(* CODESYS project OSC_MQTT.library
   Author: Peter Magnusson
   Title: MQTT Library
   Version: 1.0.0.0
   Description: Open Source CODESYS (OSC) MQTT Client library
   DefaultNamespace: OSC_MQTT
   Company: OSC

Project tree, tasks and I/O mapping:
  libraries: CmpErrors Interfaces, * (System); SysTypes Interfaces, * (System); CmpLog, 3.5.5.0 (System); Standard, 3.5.7.0 (System); CAA Types Extern, 3.5.5.0 (CAA Technical Workgroup); IoStandard, 3.5.8.0 (System); SysMem, 3.5.5.0 (System); CAA Net Base Services, 3.5.8.0 (CAA Technical Workgroup); SysTarget, 3.5.5.0 (System); CmpEventMgr, 3.5.8.0 (System); CmpApp, 3.5.8.0 (System); IoDriver Interfaces, 3.5.2.0 (System); IoDrvBase, 3.5.5.0 (System); IoDriver Parameter Interfaces, 3.5.2.0 (System); SysCpuHandling, 3.5.8.0 (System)
  MQTT/
    Enums/
      data type CLIENTSTATE
      data type MESSAGETYPE
      data type QoS
    Structs/
      data type MQTTMESSAGE
    Function Blocks/
      function block MQTTClient [ST]: _writeByte, _connect, _write, _writeString, _writeWord, _disconnect, Publish, Subscribe, _Send, _Receive, _Keepalive, Initialize
      function block MQTTPub [ST]
      function block IoDrvMQTT [ST]: FB_Init, QueryInterface, FB_Reinit, FB_Exit, Initialize, IoDrvUpdateConfiguration, IoDrvWatchdogTrigger, IoDrvGetModuleDiagnosis, IoDrvStartBusCycle, IoDrvReadInputs, IoDrvUpdateMapping, IoDrvWriteOutputs, IoDrvScanModules, IoDrvIdentify, IoDrvGetConnector, IoDrvWriteParameter, IoDrvReadParameter
    GlobalConstants/
      global variables Constants
*)

// MQTT/Enums/CLIENTSTATE
TYPE CLIENTSTATE :
(
	STOP:= 0,
	INIT,
	CONNECTING,
	CONNECTED,
	DISCONNECTING,
	DISCONNECTED,
	CLOSE,
	ERROR
);
END_TYPE

// MQTT/Enums/MESSAGETYPE
TYPE MESSAGETYPE :
(
	CONNECT 	:= 16#10,
	CONNACK 	:= 16#20,
	PUBLISH 	:= 16#30,
	PUBACK 		:= 16#40,
	SUBSCRIBE 	:= 16#80,
	SUBACK 		:= 16#90,
	UNSUBSCRIBE := 16#A0,
	UNSUBACK 	:= 16#B1,
	PINGREQ 	:= 16#C0,
	PINGRESP	:= 16#D0,
	DISCONNECT 	:= 16#E0
) BYTE;
END_TYPE

// MQTT/Enums/QoS
TYPE QoS :
(
	AtMostOnce:= 2#000,
	AtLeastOnce:= 2#010,
	ExactlyOnce:= 2#100
) BYTE;
END_TYPE

// MQTT/Structs/MQTTMESSAGE
TYPE MQTTMESSAGE :
STRUCT
	MessageType: MESSAGETYPE;
	DUP: BYTE;
	QoS: QoS;
	RetainMsg: BYTE;
	Length: BYTE;
	Payload: ARRAY[0..126] OF BYTE;
END_STRUCT
END_TYPE

// MQTT/GlobalConstants/Constants
{attribute 'qualified_only'}
VAR_GLOBAL CONSTANT	
	MQTTPROTOCOLVERSION : BYTE := BYTE#3;
	MQTT_MAX_PACKET_SIZE : BYTE := 128; //maximum packet size
	
	MQTT_MIN_KEEPALIVE : TIME := T#15S;	
	MQTT_DEFAULT_PORT : UINT := 1883;
	MQTT_MAX_CALLBACKS : INT :=3;
END_VAR

// MQTT/Function Blocks/MQTTClient
FUNCTION_BLOCK MQTTClient
VAR_INPUT
	
END_VAR
VAR_OUTPUT
	xOnline: BOOL;
	dwError: DWORD;

END_VAR
VAR
	sServerIP: STRING;
	uiPort: UINT := 1883;
	tKeepaliveInterval: TIME := T#15S;
	xEnable: BOOL;
	
	MQTT_TIMEAHEAD: TIME;
	Keepalive: TON;
	xKeepaliveEnabled: BOOL;
	xServerAlive:BOOL;

	TCPIPAddress: NBS.IP_ADDR;
	TCPClient: NBS.TCP_Client; /// FB TCP Client 
	TCPConnection: CAA.HANDLE; /// Handle to the established connection 
	TCPRead			: NBS.TCP_Read; (* FB TCP Read *)
	TCPWrite		: NBS.TCP_Write; (* FB TCP Writer *)
	RBUF: ARRAY[0..Constants.MQTT_MAX_PACKET_SIZE] OF BYTE; /// Receive Buffer
	SBUF: ARRAY[0..Constants.MQTT_MAX_PACKET_SIZE] OF BYTE; /// Send Buffer
	sLength: UINT;
	
	_nextMsgId: UINT;
	old_activate: BOOL := FALSE;
	eClientState: CLIENTSTATE;
	ePreviousClientState: CLIENTSTATE;
	cb: BYTE;
	idx1: INT;
	
	_isWriting: MESSAGETYPE; ///Command that is written.
	_hasMessage: BOOL; //has a received message to process
	msgIn: MQTTMESSAGE; //the last received message
	xSend: BOOL;
	_pConnector: POINTER TO IoConfigConnector;
	
END_VAR


Keepalive(IN:=xKeepaliveEnabled, PT:= MQTT_TIMEAHEAD);
//first case of state
IF eClientState <> ePreviousClientState THEN
	CASE eClientState OF
		CLIENTSTATE.INIT:
			{IF defined (DEBUG_MQTTCLIENT)}
			LogAdd(STD_LOGGER,'MQTTClient',UDINT_TO_DINT(LogClass.LOG_INFO),0,0,'State.INIT');
			{END_IF}
			MQTT_TIMEAHEAD:= UDINT_TO_TIME(TIME_TO_UDINT(tKeepaliveInterval) / 3 * 2);// 2/3 to be paranoid 
		CLIENTSTATE.CONNECTING:
			{IF defined (DEBUG_MQTTCLIENT)}
			LogAdd(STD_LOGGER,'MQTTClient',UDINT_TO_DINT(LogClass.LOG_INFO),0,0,'State.CONNECTING');
			{END_IF}
		CLIENTSTATE.CONNECTED:
			{IF defined (DEBUG_MQTTCLIENT)}
			LogAdd(STD_LOGGER,'MQTTClient',UDINT_TO_DINT(LogClass.LOG_INFO),0,0,'State.CONNECTED');
			{END_IF}
		CLIENTSTATE.DISCONNECTING:
			{IF defined (DEBUG_MQTTCLIENT)}
			LogAdd(STD_LOGGER,'MQTTClient',UDINT_TO_DINT(LogClass.LOG_INFO),0,0,'State.DISCONNECTING');
			{END_IF}
		CLIENTSTATE.DISCONNECTED:
			{IF defined (DEBUG_MQTTCLIENT)}
			LogAdd(STD_LOGGER,'MQTTClient',UDINT_TO_DINT(LogClass.LOG_INFO),0,0,'State.DISCONNECTED');
			{END_IF}
		CLIENTSTATE.CLOSE:		
			{IF defined (DEBUG_MQTTCLIENT)}
			LogAdd(STD_LOGGER,'MQTTClient',UDINT_TO_DINT(LogClass.LOG_INFO),0,0,'State.CLOSE');
			{END_IF}
		CLIENTSTATE.ERROR:
			{IF defined (DEBUG_MQTTCLIENT)}
			LogAdd(STD_LOGGER,'MQTTClient',UDINT_TO_DINT(LogClass.LOG_INFO),0,0,'State.ERROR');
			{END_IF}
	END_CASE
END_IF
ePreviousClientState:= eClientState;

//every time the loop is in a certain state.
CASE eClientState OF
	
	CLIENTSTATE.STOP:
		xOnline := FALSE;
		
	CLIENTSTATE.INIT:
		SysMem.SysMemSet(ADR(SBUF), 0, SIZEOF(SBUF)); //clear send buffer;
		SysMem.SysMemSet(ADR(RBUF), 0, SIZEOF(RBUF)); //clear receive buffer;
		TCPIPAddress.sAddr := sServerIP;
		xSend:=FALSE;
		dwError := 0;
		sLength:=0;
		_hasMessage:= FALSE;
		_nextMsgId := 1;
		TCPWrite(xExecute:= FALSE);
		(* The client tries to establish a connection to a mqtt server *)
		TCPClient(xEnable:= TRUE, udiTimeOut:= 0, ipAddr:= TCPIPAddress, uiPort:= uiPort, hConnection=> TCPConnection);
		
			
		IF TCPClient.xActive THEN 
			eClientState:= CLIENTSTATE.CONNECTING;
			xServerAlive:=TRUE;
			THIS^._connect();
		ELSIF TCPClient.xError THEN
			
			eClientState:= CLIENTSTATE.ERROR;
		END_IF	
	(*------------------------- *)
	

	
	CLIENTSTATE.CONNECTED:
			xKeepaliveEnabled:= TRUE;
			xOnline:= TRUE;
	(*------------------------- *)
	
	CLIENTSTATE.DISCONNECTING:
			xKeepaliveEnabled:=FALSE;
			IF NOT xSend THEN
				eClientState:= DISCONNECTED;
			END_IF
	(*------------------------- *)	
	
	CLIENTSTATE.DISCONNECTED:		
		//logger('disconnected');
		xKeepaliveEnabled:=FALSE;
		eClientState:= CLOSE;
	(*------------------------- *)
	
	CLIENTSTATE.ERROR:
		xSend:=FALSE;
		TCPClient(xEnable := FALSE);
		eCLientState:= CLOSE;
		
	(*------------------------- *)
	
	CLIENTSTATE.CLOSE:		
		//logger('close');
		xServerAlive:=FALSE;
		xKeepaliveEnabled:=FALSE;
		old_activate := FALSE;
		xOnline:= FALSE;
		
		TCPWrite(xExecute:= FALSE);
		TCPRead(xEnable:=FALSE);
		TCPClient(xEnable:= FALSE);
		
		eClientState := CLIENTSTATE.STOP;
		
		
		
	(*------------------------- *)
	
END_CASE




//IPC1(IP:= DWORD#0, PORT:= WORD#0 , TIME_OUT:= TIMEOUT, IP_C:= IP_C1, S_BUF:= S_BUF1, R_BUF:= R_BUF1); (* MQTT Connection *)




IF NOT old_activate AND xEnable THEN
	eClientState := INIT;
	old_activate:= TRUE;
END_IF

IF NOT xEnable AND old_activate THEN
	{IF defined (DEBUG_MQTTCLIENT)}
	LogAdd(STD_LOGGER,'MQTTClient',UDINT_TO_DINT(LogClass.LOG_INFO),0,0,'Falling flank of xConnect ');
	{END_IF}
	THIS^._disconnect();
	old_activate:= FALSE;
END_IF

IF xSend AND TCPConnection = CAA.gc_hINVALID THEN
	xSend:= FALSE;
	IF eClientState <= CLIENTSTATE.DISCONNECTED THEN
		eClientState:= CLIENTSTATE.DISCONNECTED;
	END_IF
	
END_IF


IF TCPClient.xEnable AND TCPClient.xActive AND TCPClient.hConnection <> CAA.gc_hINVALID THEN
	THIS^._Keepalive();
	THIS^._Send();
	THIS^._Receive();
END_IF

METHOD PRIVATE _writeByte : INT
VAR_IN_OUT
	pos: UINT;
END_VAR
VAR_INPUT
	b: BYTE;
	pBuf: POINTER TO ARRAY[0..Constants.MQTT_MAX_PACKET_SIZE] OF BYTE;
END_VAR
//Add to current position according to size
pBuf^[pos]:= b;
//increase size
pos:= pos +1;
END_METHOD

METHOD PRIVATE _connect : BOOL
VAR_INPUT

END_VAR
VAR
	name: WSTRING:="01234567890123456789";
	dwId: DWORD;
	id: STRING;
	v: BYTE;
	w: UINT;
	length: UINT;
	MAX_NAME_LENGTH: UDINT := 20;
END_VAR

IF TCPClient.xActive THEN
		
	SysTarget.SysTargetGetNodeName(ADR(name), ADR(MAX_NAME_LENGTH));
	SysTarget.SysTargetGetId(ADR(dwId));
	id := CONCAT('mqttio/', WSTRING_TO_STRING(name));
	id := CONCAT(id, '-');
	id := CONCAT(id, DWORD_TO_STRING(dwId));
	
	 

	// {0x00,0x06,'M','Q','I','s','d','p',MQTTPROTOCOLVERSION};
	//leave room in the buffer for header and variable field length field
	length:=2;
	//start adding
	_writeByte(pos:=length, b:=16#0, pBuf := ADR(SBUF));
	_writeByte(pos:=length, b:=16#6, pBuf := ADR(SBUF));
	_writeString(pos:=length, msg:='MQIsdp');
	_writeByte(pos:=length, b:=Constants.MQTTPROTOCOLVERSION, pBuf := ADR(SBUF));
	
	//connect flags
	v := 16#2;//no will topic
	_writeByte(pos:=length, b:=v, pBuf := ADR(SBUF));
	
	//Keep Alive Timer
	_writeWord(pos:=length, w:= TIME_TO_WORD(tKeepaliveInterval/1000),  pBuf := ADR(SBUF)); 
	
	//client id length
	w:= INT_TO_UINT(LEN(id));
	_writeWord(pos:=length, w:=w,  pBuf := ADR(SBUF));
	//client id
	_writeString(pos:=length, msg:=id);
	_write(MESSAGETYPE.CONNECT, length);

END_IF
END_METHOD

METHOD PRIVATE _write : BOOL
VAR_INPUT
	header: MESSAGETYPE;
	length: UINT;
END_VAR
VAR
	len: BYTE;
END_VAR
IF TCPClient.xActive THEN	
	{IF defined (DEBUG_MQTTCLIENT)}
	LogAdd(STD_LOGGER,'MQTTClient',UDINT_TO_DINT(LogClass.LOG_INFO),0,0,CONCAT('Writing msg:', BYTE_TO_STRING(header) ));
	{END_IF}
	_isWriting:= header;
	len:= UINT_TO_BYTE(length);
	SBUF[0]:= header;
	IF len >= 2 THEN
		SBUF[1]:= len -2;
	ELSE
		SBUF[1]:= 0;
	END_IF
	
	IF(length<2) THEN
		length:= 2;
	END_IF
	sLength:= length;
	xSend:= TRUE;
END_IF
END_METHOD

METHOD PRIVATE _writeString
VAR_IN_OUT
	pos: UINT;
END_VAR
VAR_INPUT
	msg: STRING;
	
END_VAR

VAR
	ps : POINTER TO BYTE;
	end: UINT;
	i: UINT;
	length: UINT;
END_VAR
ps := ADR(msg);
length := INT_TO_UINT(LEN(msg));
end := MIN(pos + length, SIZEOF(SBUF));
IF end > 0 THEN end := end -1; END_IF;
FOR i := pos TO end DO
	SBUF[i] := ps^;
	ps := ps + 1;
END_FOR;
pos:=pos + length;
END_METHOD

METHOD PRIVATE _writeWord : INT
VAR_IN_OUT
	pos: UINT;
END_VAR
VAR_INPUT
	w: WORD;
	pBuf: POINTER TO ARRAY[0..Constants.MQTT_MAX_PACKET_SIZE] OF BYTE;
END_VAR
VAR
	v: BYTE;
	length: UINT;
END_VAR
length:= pos;
v:= UINT_TO_BYTE(SHR(w, 8));
_writeByte(pos:=length, b:=v, pBuf:=pBuf );
v:= UINT_TO_BYTE(w AND 16#FF);
_writeByte(pos:=length, b:=v, pBuf := pBuf); 
pos:= length;
END_METHOD

METHOD PRIVATE _disconnect
VAR_INPUT
END_VAR

VAR
	
END_VAR
{IF defined (DEBUG_MQTTCLIENT)}
LogAdd(STD_LOGGER,'MQTTClient',UDINT_TO_DINT(LogClass.LOG_INFO),0,0,'Calling _Disconnect');
{END_IF}
SysMem.SysMemSet(ADR(SBUF), 0, Constants.MQTT_MAX_PACKET_SIZE); //clear send buffer;
THIS^._write(MESSAGETYPE.DISCONNECT, 0);
eCLIENTSTATE:= CLIENTSTATE.DISCONNECTING;
END_METHOD

METHOD Publish
VAR_INPUT
	sTopic: STRING;
	sValue: STRING;
	xExecute: BOOL;
	bQos: BYTE;
	xRetain:BOOL;
END_VAR
VAR_OUTPUT
	xDone:BOOL;
END_VAR
VAR
	length: UINT;
	xBusyPublishing:BOOL; //will be set if publishing
	bBuf : ARRAY[0..Constants.MQTT_MAX_PACKET_SIZE] OF BYTE; /// Send Buffer
END_VAR

IF xExecute AND NOT xBusyPublishing THEN //Rising flank
	IF TCPClient.xActive THEN
		{IF defined (DEBUG_MQTTCLIENT)}
		LogAdd(STD_LOGGER,'MQTTClient',UDINT_TO_DINT(LogClass.LOG_INFO),0,0,'Publishing');
		{END_IF}
		xDone:=FALSE;
		xBusyPublishing:=TRUE;
		//sTopic := concat(sTopicPrefix, sTopic);
		length:= 2;//starting position in the buffer
		_writeWord(pos:=length, w:= INT_TO_UINT(LEN(sTopic)), pBuf := ADR(bBuf));
		_writeString(pos:=length, msg:=sTopic);
		IF bQos > 0 THEN //only send msg id if needed.
			_writeWord(pos:=length, w:= _nextMsgId, pBuf := ADR(SBUF));
		END_IF
		_writeString(pos:=length, msg:=sValue);
		_write(MESSAGETYPE.PUBLISH, length);
	END_IF
ELSIF NOT xExecute AND xBusyPublishing THEN //falling flank
	{IF defined (DEBUG_MQTTCLIENT)}
	LogAdd(STD_LOGGER,'MQTTClient',UDINT_TO_DINT(LogClass.LOG_INFO),0,0,'Publishing falling');
	{END_IF}
	xDone:=FALSE;
	xBusyPublishing:=FALSE;
ELSIF xExecute AND xBusyPublishing THEN //steady high
	//TODO:Wait for PUBACK if QoS >0
	IF NOT xSend THEN
		{IF defined (DEBUG_MQTTCLIENT)}
		LogAdd(STD_LOGGER,'MQTTClient',UDINT_TO_DINT(LogClass.LOG_INFO),0,0,'Publishing Done');
		{END_IF}
		xDone:=TRUE;
	END_IF
END_IF
END_METHOD

METHOD Subscribe : BOOL
VAR_INPUT
	sTopic: STRING;
	//pfbCallback: POINTER TO IMqttMessage;
END_VAR

VAR
	length: UINT;
END_VAR
//Save callback for later and send subscribe message
//m_Subscriptions.AddSub(sTopic:=sTopic, pfbCallback:=pfbCallback);

//leave room in the buffer for header and variable field length field
length:=2;

//topic and length of topic
_writeWord(pos:=length, INT_TO_UINT(LEN(sTopic)), pBuf := ADR(SBUF));
_writeString(pos:=length, msg:=sTopic);

//requested qos
_writeByte(pos:=length, b:=0, pBuf := ADR(SBUF));

_write(MESSAGETYPE.SUBSCRIBE, length);
END_METHOD

METHOD PRIVATE _Send
VAR_INPUT
END_VAR
IF xSend THEN
	

{IF defined (DEBUG_MQTTCLIENT)}
LogAdd(STD_LOGGER,'MQTTClient',UDINT_TO_DINT(LogClass.LOG_INFO),0,0,'Sending...');
{END_IF}
TCPWrite(xExecute:= TRUE, udiTimeOut:= 0, hConnection:= TCPConnection, szSize:= sLength, pData:= ADR(SBUF));
IF TCPWrite.xDone THEN 
	_nextMsgId:= _nextMsgId +1;				
	TCPWrite(xExecute:= FALSE);	
	xSend:= FALSE;
	sLength:= 0;		
	{IF defined (DEBUG_MQTTCLIENT)}
	LogAdd(STD_LOGGER,'MQTTClient',UDINT_TO_DINT(LogClass.LOG_INFO),0,0,'Sent');
	{END_IF}	
ELSIF TCPWrite.xError THEN
	//eCLIENTSTATE := CLIENTSTATE.ERROR;
	TCPWrite(xExecute:=FALSE);
	xSend:= FALSE;
	sLength:=0;
	{IF defined (DEBUG_MQTTCLIENT)}
	LogAdd(STD_LOGGER,'MQTTClient',UDINT_TO_DINT(LogClass.LOG_INFO),0,0,'Error Sending');
	{END_IF}
END_IF
IF _isWriting = MESSAGETYPE.DISCONNECT THEN
	eClientState := CLIENTSTATE.DISCONNECTED;
	xSend:=FALSE;
	{IF defined (DEBUG_MQTTCLIENT)}
	LogAdd(STD_LOGGER,'MQTTClient',UDINT_TO_DINT(LogClass.LOG_INFO),0,0,'Send Disconnect');
	{END_IF}
END_IF

END_IF
END_METHOD

METHOD PRIVATE _Receive
VAR_INPUT
END_VAR
TCPRead(xEnable:= TRUE, hConnection:= TCPConnection, szSize:= Constants.MQTT_MAX_PACKET_SIZE, pData:= ADR(RBUF));
IF TCPRead.xReady AND TCPRead.szCount > 0 THEN
	msgIn.MessageType := RBUF[0] AND 16#F0; //mask of first half
	msgIn.DUP := RBUF[0] AND 16#08;
	msgIn.QoS := RBUF[0] AND 16#06;
	msgIn.RetainMsg := RBUF[0] AND 1;
	msgIn.Length := RBUF[1]; //remaining length;
	SysMem.SysMemCpy(ADR(msgIn.Payload[0]), ADR(RBUF[2]), msgIn.Length);
	_hasMessage := TRUE;
	{IF defined (DEBUG_MQTTCLIENT)}
	LogAdd(STD_LOGGER,'MQTTClient',UDINT_TO_DINT(LogClass.LOG_INFO),0,0,CONCAT('Received:', BYTE_TO_STRING(msgIn.MessageType)));
	{END_IF}
ELSIF TCPRead.xError THEN
	eClientState := CLIENTSTATE.ERROR;
	{IF defined (DEBUG_MQTTCLIENT)}
	LogAdd(STD_LOGGER,'MQTTClient',UDINT_TO_DINT(LogClass.LOG_INFO),0,0,'Receive Error');
	{END_IF}
END_IF




IF _hasMessage THEN
//logger('hasMessage');	
	CASE _isWriting OF
		MESSAGETYPE.CONNECT:
			IF msgIn.MessageType = MESSAGETYPE.CONNACK THEN
				IF msgIn.Payload[1] = 0 THEN //connection accepted
					eClientState:= CONNECTED; 
					
				ELSE
					{IF defined (DEBUG_MQTTCLIENT)}
					LogAdd(STD_LOGGER,'MQTTClient',UDINT_TO_DINT(LogClass.LOG_INFO),0,0,'Could not authenticate');
					{END_IF}
					eClientState:= CLOSE;	
				END_IF
			END_IF
		(*----------------------------*)
		
		MESSAGETYPE.SUBSCRIBE:
			IF msgIn.MessageType = MESSAGETYPE.SUBACK THEN
				{IF defined (DEBUG_MQTTCLIENT)}
				LogAdd(STD_LOGGER,'MQTTClient',UDINT_TO_DINT(LogClass.LOG_INFO),0,0,'SUBACK');
				{END_IF}
			ELSE
				{IF defined (DEBUG_MQTTCLIENT)}
				LogAdd(STD_LOGGER,'MQTTClient',UDINT_TO_DINT(LogClass.LOG_INFO),0,0,'SUBACK EXPECTED BUT NOT RECEIVED');
				{END_IF}	
			END_IF
			
		(*----------------------------*)
		
		MESSAGETYPE.PINGREQ:
			IF msgIn.MessageType = MESSAGETYPE.PINGRESP THEN
				//server alive
				{IF defined (DEBUG_MQTTCLIENT)}
				LogAdd(STD_LOGGER,'MQTTClient',UDINT_TO_DINT(LogClass.LOG_INFO),0,0,'PINGRESP');
				{END_IF}
				xServerAlive:=TRUE;
			END_IF 
		(*----------------------------*)
		
	
	END_CASE
_hasMessage:= FALSE; //message is dealt with
END_IF
END_METHOD

METHOD PRIVATE _Keepalive
VAR_INPUT
END_VAR
//keepalive triggered
IF Keepalive.Q THEN
	xKeepaliveEnabled:= FALSE;
	IF NOT xServerAlive THEN
		//SOMETHING BAD HAPPENED
		{IF defined (DEBUG_MQTTCLIENT)}
		LogAdd(STD_LOGGER,'MQTTClient',UDINT_TO_DINT(LogClass.LOG_INFO),0,0,'Something bad happened with connection');
		{END_IF}
		eClientState:= CLOSE;
	ELSE
		//check if server is alive.
		xServerAlive:=FALSE;
		{IF defined (DEBUG_MQTTCLIENT)}
		LogAdd(STD_LOGGER,'MQTTClient',UDINT_TO_DINT(LogClass.LOG_INFO),0,0,'PINGREQ');
		{END_IF}
		_write(MESSAGETYPE.PINGREQ, 0);
	END_IF
END_IF
END_METHOD

METHOD Initialize : UDINT
VAR_INPUT
	wModuleType : UINT;
	dwInstance : UDINT;
	pConnector : POINTER TO IoConfigConnector;
END_VAR
VAR
	pParam: POINTER TO IoConfigParameter;		
	udiResult: UDINT;
END_VAR

pParam := ConfigGetParameter(_pConnector, 1);
IF pParam <> 0 THEN
	_byHardwareAddress := IoStandard.ConfigGetParameter(pParam, ADR(udiResult));
END_IF
END_METHOD

END_FUNCTION_BLOCK

// MQTT/Function Blocks/MQTTPub
FUNCTION_BLOCK MQTTPub
VAR_INPUT
	pClient		:POINTER TO MQTTClient;
	sTopic		:STRING;
	sValue		:STRING;
	xExecute	:BOOL;
END_VAR
	
VAR_OUTPUT
	xDone		:BOOL;
END_VAR
VAR
	
END_VAR

IF xExecute THEN
	pClient^.Publish(sTopic:=sTopic, sValue:=sValue, bQos:=0, xRetain:=FALSE, xExecute:=TRUE, xDone => xDone);
END_IF

END_FUNCTION_BLOCK

// MQTT/Function Blocks/IoDrvMQTT
FUNCTION_BLOCK IoDrvMQTT EXTENDS IoDrvBase IMPLEMENTS ICmpIoDrvParameter
VAR_INPUT
END_VAR
VAR_OUTPUT
	
END_VAR
VAR CONSTANT
	CLASSID_CCmpIoDrvTemplate : DWORD := 16#0000FF02; //TODO
	_IIoDrv : ICmpIoDrv;
	_IIoDrvParameter : ICmpIoDrvParameter;
	_xBackGroundDiagStarted : BOOL;
	_bDeactivated : BOOL;
	Client: MQTTClient;
END_VAR

VAR
END_VAR

{attribute 'conditionalshow'}
METHOD FB_Init : BOOL
VAR_INPUT
	bInitRetains	: BOOL;
	bInCopyCode	: BOOL;
END_VAR
VAR
	Result : UDINT;
END_VAR
FB_Init_Count := FB_Init_Count + 1;

m_Info.szDriverName := 'IoDrvMQTT';
m_Info.szVendorName := 'Open Source CODESYS (OSC)';
m_Info.szDeviceName := 'MQTT';
m_Info.wModuleType := 501;

_IIoDrv := THIS^;
_IIoDrvParameter := THIS^;

m_IBaseItf := THIS^;
m_hInterface := IoMgrRegisterInstance2(CLASSID_CCmpIoDrvTemplate, m_IBaseItf, ADR(Result));
FB_Init := TRUE;
END_METHOD

{attribute 'conditionalshow'}
METHOD QueryInterface : POINTER TO POINTER TO BYTE
VAR_INPUT
	(* InterfaceID *)
	iid	: DWORD;
	pResult	: POINTER TO UDINT;
END_VAR
QueryInterface_Count := QueryInterface_Count + 1;
IF iid = ITFID_ICmpIoDrv THEN
	QueryInterface := ADR(_IIoDrv);
	AddRef();
	IF (pResult <> 0) THEN
		pResult^ := Errors.ERR_OK;
	END_IF
	RETURN;	
ELSIF iid = ITFID_ICmpIoDrvParameter THEN
	QueryInterface := ADR(_IIoDrvParameter);
	AddRef();
	IF (pResult <> 0) THEN
		pResult^ := Errors.ERR_OK;
	END_IF	
	RETURN;	
ELSE
	QueryInterface := SUPER^.QueryInterface(iid, pResult);
END_IF
END_METHOD

{attribute 'conditionalshow'}
METHOD FB_Reinit : BOOL
FB_Reinit_Count := FB_Reinit_Count + 1;
FB_Reinit := TRUE;
END_METHOD

{attribute 'conditionalshow'}
METHOD FB_Exit : BOOL
VAR_INPUT
	bInCopyCode	: BOOL;
END_VAR
FB_Exit_Count := FB_Exit_Count + 1;
FB_Exit := TRUE;
END_METHOD

{attribute 'conditionalshow'}
METHOD Initialize : UDINT
VAR_INPUT
	wModuleType : UINT;
	dwInstance : UDINT;
	pConnector : POINTER TO IoConfigConnector; 
END_VAR
Initialize_Count := Initialize_Count + 1;

m_wModuleType := wModuleType;
m_dwInstance := dwInstance;
m_Info.wModuleType := wModuleType;

Client.Initialize(wModuleType, dwInstance, pConnector);

Initialize := Errors.ERR_OK;
END_METHOD

{attribute 'conditionalshow'}
METHOD IoDrvUpdateConfiguration : UDINT
VAR_INPUT
	pConnectorList	: POINTER TO IoConfigConnector;
	nCount	: DINT;
END_VAR

VAR
	pParameter : POINTER TO IoConfigParameter;	
	pChild : POINTER TO IoConfigConnector;	
	pstConnectorVendorName : POINTER TO STRING;
	pstConnectorDeviceName : POINTER TO STRING;
	dwTest : POINTER TO DWORD;
	Result : RTS_IEC_RESULT;
END_VAR
IoDrvUpdateConfiguration_Count := IoDrvUpdateConfiguration_Count + 1;
IoDrvUpdateConfiguration := Errors.ERR_OK;

IF (pConnectorList = 0) THEN
	// Reset application
	// TODO: Free ressources
	RETURN;
END_IF

m_pConnector := IoMgrConfigGetConnector(pConnectorList, ADR(nCount), m_wModuleType, m_dwInstance);

IF m_pConnector = 0 THEN
	IoDrvUpdateConfiguration := ERRORS.ERR_PARAMETER;
	RETURN;
END_IF

//check if device is enabled in the device tree
IF (m_pConnector^.dwFlags AND ConnectorFlags.CF_ENABLE) = 0 THEN
	_bDeactivated := TRUE;
	IoDrvUpdateConfiguration := Errors.ERR_OK;
	RETURN;
END_IF

IF m_pConnector^.hIoDrv = 0 THEN
	m_pConnector^.hIoDrv := m_hInterface;
	m_pConnector^.pFather^.hIoDrv := m_hInterface;
	
	{IF defined (pou:IoMgrConfigSetDiagnosis)}
	IoMgrConfigSetDiagnosis(m_pConnector,
							ConnectorFlags.CF_DRIVER_AVAILABLE OR
							ConnectorFlags.CF_CONNECTOR_FOUND OR
							ConnectorFlags.CF_CONNECTOR_CONFIGURED OR
							ConnectorFlags.CF_CONNECTOR_ACTIVE);
	{END_IF}
	
	{IF defined (pou:IoMgrConfigSetDiagnosis)}
	IoMgrConfigSetDiagnosis(m_pConnector^.pFather,
							ConnectorFlags.CF_DRIVER_AVAILABLE OR
							ConnectorFlags.CF_CONNECTOR_FOUND OR
							ConnectorFlags.CF_CONNECTOR_CONFIGURED OR
							ConnectorFlags.CF_CONNECTOR_ACTIVE);
	{END_IF}

	{IF defined (pou:IoMgrSetDriverProperties)}			
		IoMgrSetDriverProperties(m_hInterface, DRVPROP_CONSISTENCY OR DRVPROP_BACKGROUND_GETDIAG);
		//Note: background diagnosis property flag is optional (supported with 3.5.1.0 runtime)
	{END_IF}										

	//Setup I/O area
	pParameter := IoMgrConfigGetParameter(m_pConnector, 1000);		(* inputs *)
	IF (pParameter <> 0) THEN
		pParameter^.dwDriverSpecific := 0;					(* Device offset 0 *)
	END_IF
	pParameter := IoMgrConfigGetParameter(m_pConnector, 2000);		(* outputs *)
	IF (pParameter <> 0) THEN
		pParameter^.dwDriverSpecific := 0;					(* Device offset 0 *)
	END_IF
	
	//Go through all childs of the device
	pChild := IoMgrConfigGetFirstChild(m_pConnector, ADR(nCount), m_pConnector);
	WHILE (pChild <> 0) DO
		IF (pChild^.dwFlags AND ConnectorFlags.CF_ENABLE) <> 0 THEN
			pChild^.hIoDrv := m_hInterface;	
			{IF defined (pou:IoMgrConfigSetDiagnosis)}
			IoMgrConfigSetDiagnosis(pChild,
									ConnectorFlags.CF_DRIVER_AVAILABLE OR
									ConnectorFlags.CF_CONNECTOR_FOUND OR
									ConnectorFlags.CF_CONNECTOR_CONFIGURED OR
									ConnectorFlags.CF_CONNECTOR_ACTIVE);
			{END_IF}
		END_IF
		pChild := IoMgrConfigGetNextChild(pChild, ADR(nCount), m_pConnector);
	END_WHILE
END_IF
END_METHOD

{attribute 'conditionalshow'}
METHOD IoDrvWatchdogTrigger : UDINT
VAR_INPUT
	pConnector	: POINTER TO IoConfigConnector;
END_VAR
IoDrvWatchdogTrigger_Count := IoDrvWatchdogTrigger_Count + 1;
IoDrvWatchdogTrigger := Errors.ERR_OK;
END_METHOD

{attribute 'conditionalshow'}
METHOD IoDrvGetModuleDiagnosis : UDINT
VAR_INPUT
	pConnector	: POINTER TO IoConfigConnector;
END_VAR
IF pConnector = 0 THEN
	//we are called from the background task
	_xBackGroundDiagStarted := TRUE;
END_IF

//Todo: update connectorflags if something changed

IoDrvGetModuleDiagnosis_Count := IoDrvGetModuleDiagnosis_Count + 1;
IoDrvGetModuleDiagnosis := Errors.ERR_NOTIMPLEMENTED;
END_METHOD

{attribute 'conditionalshow'}
METHOD IoDrvStartBusCycle : UDINT
VAR_INPUT
	pConnector	: POINTER TO IoConfigConnector;
END_VAR
IoDrvStartBusCycle_Count := IoDrvStartBusCycle_Count + 1;

//if background diagnosis is not active call IoDrvGetModuleDiagnosis; normally it will be called by the runtime if DRVPROP_BACKGROUND_GETDIAG is set
IF NOT _xBackGroundDiagStarted THEN
	IoDrvGetModuleDiagnosis(m_pConnector); //DRVPROP_BACKGROUND_GETDIAG not set or runtime version < V3.5.1.0
END_IF

//optional: call IoDrvWatchdogTrigger or set driver property DRVPROP_WATCHDOG in UpdateConfiguration
IoDrvWatchdogTrigger(pConnector);

IF NOT _bDeactivated THEN
	//Check subscriptions
	Client.AfterReadInputs();
	
	//Publish
	Client.BeforeWriteOutputs();
END_IF

IoDrvStartBusCycle := Errors.ERR_OK;
END_METHOD

{attribute 'conditionalshow'}
METHOD IoDrvReadInputs : UDINT
VAR_INPUT
	pConnectorMapList	: POINTER TO IoConfigConnectorMap;
	nCount	: DINT;
END_VAR
VAR
	i,j : DINT;
	wSize : WORD;
	pbyIecAddress : POINTER TO BYTE;
	bySrcValue : BYTE;
	bySrcMask : BYTE;
	wSrcIndex : WORD;	
	wDestIndex : WORD;	
END_VAR
IoDrvReadInputs_Count := IoDrvReadInputs_Count + 1;

IF pConnectorMapList = 0 OR nCount = 0 THEN
	IoDrvReadInputs := Errors.ERR_PARAMETER;
	RETURN;
END_IF

FOR i:=0 TO nCount - 1 DO
	IF (pConnectorMapList[i].dwNumOfChannels = 0) THEN
		CONTINUE;
	END_IF
	FOR j:= 0 TO UDINT_TO_UINT(pConnectorMapList[i].dwNumOfChannels) - 1 DO		
		pbyIecAddress := pConnectorMapList[i].pChannelMapList[j].pbyIecAddress;
		wDestIndex := pConnectorMapList[i].pChannelMapList[j].wIecAddressBitOffset / 8;
		IF (pConnectorMapList[i].pChannelMapList[j].wSize = 1) THEN
			IF (PiFace.byIn AND SHL(BYTE#1, pConnectorMapList[i].pChannelMapList[j].wParameterBitOffset MOD 8)) <> 0 THEN
			{IF defined (pou:SysCpuSetBit2)}
				SysCpuSetBit2(ADR(pbyIecAddress[wDestIndex]), pConnectorMapList[i].pChannelMapList[j].wIecAddressBitOffset MOD 8);			
    		{ELSE}    
				SysCpuSetBit(ADR(pbyIecAddress[wDestIndex]), pConnectorMapList[i].pChannelMapList[j].wIecAddressBitOffset MOD 8);			
    		{END_IF}    
			ELSE
			{IF defined (pou:SysCpuResetBit2)}
				SysCpuResetBit2(ADR(pbyIecAddress[wDestIndex]), pConnectorMapList[i].pChannelMapList[j].wIecAddressBitOffset MOD 8);			
    		{ELSE}    
				SysCpuResetBit(ADR(pbyIecAddress[wDestIndex]), pConnectorMapList[i].pChannelMapList[j].wIecAddressBitOffset MOD 8);			
    		{END_IF}    
			END_IF 			 			
		ELSIF pConnectorMapList[i].pChannelMapList[j].wSize = 8 THEN
			pbyIecAddress[wDestIndex] := PiFace.byIn;
		END_IF
	END_FOR
END_FOR

IoDrvReadInputs := Errors.ERR_OK;
END_METHOD

{attribute 'conditionalshow'}
METHOD IoDrvUpdateMapping : UDINT
VAR_INPUT
	pTaskMapList	: POINTER TO IoDriver_Interfaces.IoConfigTaskMap;
	nCount	: DINT;
END_VAR
IoDrvUpdateMapping_Count := IoDrvUpdateMapping_Count + 1;

IF (pTaskMapList = 0) THEN
	IoDrvUpdateMapping := Errors.ERR_PARAMETER;
	RETURN;
END_IF

IoDrvUpdateMapping := Errors.ERR_OK;
END_METHOD

{attribute 'conditionalshow'}
METHOD IoDrvWriteOutputs : UDINT
VAR_INPUT
	pConnectorMapList	: POINTER TO IoDriver_Interfaces.IoConfigConnectorMap;
	nCount	: DINT;
END_VAR
VAR
	i,j : DINT;
	wSize : WORD;
	pbyIecAddress : POINTER TO BYTE;
	bySrcValue : BYTE;
	wSrcIndex : WORD;	
	bySrcMask : BYTE;
	wDestIndex : WORD;	
END_VAR
IoDrvWriteOutputs_Count := IoDrvWriteOutputs_Count + 1;

IF pConnectorMapList = 0 OR nCount = 0 THEN
	IoDrvWriteOutputs := Errors.ERR_PARAMETER;
	RETURN;
END_IF

FOR i:=0 TO nCount - 1 DO
	IF (pConnectorMapList[i].dwNumOfChannels = 0) THEN
		CONTINUE;
	END_IF
	FOR j:= 0 TO UDINT_TO_UINT(pConnectorMapList[i].dwNumOfChannels) - 1 DO
		wSrcIndex := pConnectorMapList[i].pChannelMapList[j].wIecAddressBitOffset / 8; 
		pbyIecAddress := pConnectorMapList[i].pChannelMapList[j].pbyIecAddress;			

		IF pConnectorMapList[i].pChannelMapList[j].wSize = 1 THEN
			bySrcValue := pbyIecAddress[wSrcIndex];
					
			IF (pbyIecAddress[wSrcIndex] AND SHL(BYTE#1, pConnectorMapList[i].pChannelMapList[j].wIecAddressBitOffset MOD 8)) <> 0 THEN
			{IF defined (pou:SysCpuSetBit2)}
				SysCpuSetBit2(ADR(PiFace.byOut), pConnectorMapList[i].pChannelMapList[j].wParameterBitOffset MOD 8);			
    		{ELSE}    
				SysCpuSetBit(ADR(PiFace.byOut), pConnectorMapList[i].pChannelMapList[j].wParameterBitOffset MOD 8);			
    		{END_IF}    
			ELSE
			{IF defined (pou:SysCpuResetBit2)}
				SysCpuResetBit2(ADR(PiFace.byOut), pConnectorMapList[i].pChannelMapList[j].wParameterBitOffset MOD 8);				
    		{ELSE}    
				SysCpuResetBit(ADR(PiFace.byOut), pConnectorMapList[i].pChannelMapList[j].wParameterBitOffset MOD 8);				
    		{END_IF}    
			END_IF			
		ELSIF pConnectorMapList[i].pChannelMapList[j].wSize = 8 THEN
			PiFace.byOut := pbyIecAddress[wSrcIndex];
		END_IF
	END_FOR
END_FOR

IoDrvWriteOutputs := Errors.ERR_OK;
END_METHOD

{attribute 'conditionalshow'}
METHOD IoDrvScanModules : UDINT
VAR_INPUT
	pConnector	: POINTER TO IoConfigConnector;
	ppConnectorList	: POINTER TO POINTER TO IoConfigConnector;
	pnCount	: POINTER TO DINT;
END_VAR
IoDrvScanModules_Count := IoDrvScanModules_Count + 1;
IoDrvScanModules := Errors.ERR_NOTIMPLEMENTED;
END_METHOD

{attribute 'conditionalshow'}
METHOD IoDrvIdentify : UDINT
VAR_INPUT
	pConnector	: POINTER TO IoConfigConnector;
END_VAR
IoDrvIdentify_Count := IoDrvIdentify_Count + 1;
IoDrvIdentify := Errors.ERR_NOTIMPLEMENTED;
END_METHOD

{attribute 'conditionalshow'}
METHOD IoDrvGetConnector : POINTER TO IoConfigConnector
VAR_INPUT
	pResult : POINTER TO RTS_IEC_RESULT;
END_VAR
VAR
END_VAR
IF m_pConnector = 0 THEN
	IF pResult <> 0 THEN
		pResult^ := Errors.ERR_FAILED;
	END_IF
	IoDrvGetConnector := 0;	
	RETURN;
END_IF
IF pResult <> 0 THEN
	pResult^ := Errors.ERR_OK;
END_IF
IoDrvGetConnector := m_pConnector;
END_METHOD

{attribute 'conditionalshow'}
METHOD IoDrvWriteParameter : UDINT
VAR_INPUT
	pConnector	: POINTER TO IIoDrvParameter.IoConfigConnector;
	pParameter	: POINTER TO IIoDrvParameter.IoConfigParameter;
	pData	: POINTER TO BYTE;
	dwBitSize	: DWORD;
	dwBitOffset	: DWORD;
END_VAR
IF pConnector = 0 OR pParameter = 0 OR pData = 0 THEN
	IoDrvWriteParameter := Errors.ERR_PARAMETER;
	RETURN;	
END_IF

IoDrvWriteParameter := Errors.ERR_FAILED;
END_METHOD

{attribute 'conditionalshow'}
METHOD IoDrvReadParameter : UDINT
VAR_INPUT
	pConnector	: POINTER TO IIoDrvParameter.IoConfigConnector;
	pParameter	: POINTER TO IIoDrvParameter.IoConfigParameter;
	pData	: POINTER TO BYTE;
	dwBitSize	: DWORD;
	dwBitOffset	: DWORD;
END_VAR
IF 	pConnector = 0 OR pParameter = 0 OR pData = 0 THEN
	IoDrvReadParameter := Errors.ERR_PARAMETER;
	RETURN;	
END_IF

// All standard parameters of our device are handled by the IO-manager!
IoDrvReadParameter := Errors.ERR_FAILED;
END_METHOD

END_FUNCTION_BLOCK
